(* CODESYS project AxisTest.project

Project tree, tasks and I/O mapping:
  Device : AC801-0221-U0R0, Shenzhen Inovance Technology Co., Ltd., version 3.5.11.50
    application Application
      libraries: Standard, * (System)
      task MainTask (cyclic, interval 4 ms, priority 2) calls nothing
      task ETHERCAT_C (cyclic, interval 4000 µs, priority 0) calls ETHERCAT_C.EtherCAT_Task, PLC_PRG
      program PLC_PRG [ST]
      DifferentialMonitor
      trace Trace (task ETHERCAT_C): PLC_PRG.adFbPos[0], PLC_PRG.adFbPos[1], PLC_PRG.adFbPos[2], PLC_PRG.adFbPos[3], PLC_PRG.lResult
      Symbols
    HardWare Configuration
    Network Configuration
      EtherCAT Config
    Device Diagnosis
    Resources List
    ConfigStorage
    SoftMotion General Axis Pool
    MODBUS_TCP : ModbusTCP本地从站, inovance, version 00.00.00.10
    HwConfiguratioinDevice : SystemConfig, Inovance, version 00.00.00.10
        settings: NetworkConfigArray.NetworkConfigArray.BusType = 10; NetworkConfigArray.NetworkConfigArray.RackSum = 1; NetworkConfigArray.NetworkConfigArray.HardwareConfigArray.HardwareConfigArray.RackNo = 1
    ETHERCAT_C : EtherCAT Master SoftMotion, 3S - Smart Software Solutions GmbH, version 3.5.11.10
        settings:  = 0; NetworkName = 'enp3s0'; SelectNetworkByName = TRUE; DisableTaskGeneration = True
      InoSV630N_3 : SV630_1Axis_03715, Inovance, order no. InoSV630N, version Revision=16#00010000
          settings: Number of Outputs = 6; Number of Inputs = 10; Number of Infos about Outputs = 6; Number of Infos about Inputs = 10; StationAlias = 0; Sync.Length = 18; Sync.Length = 32; FMMU.Length = 18; FMMU.Length = 32; AutoUpdate = False; DC sync0 cycletime = 4000; DC sync1 cycletime = 4000; Number of SDO = 10; Homing method.Index = 16#6098; Homing method.Subindex = 16#00; Homing method.Value = 1; Homing method.Size = 8; Homing method.AbortIfError = FALSE; Homing method.JumpToLine = FALSE; Homing method.Line = 0; Homing method.CompleteAccess = FALSE; Actual Position Calculation Method.Index = 16#60E6; Actual Position Calculation Method.Subindex = 16#00; Actual Position Calculation Method.Value = 0; Actual Position Calculation Method.Size = 8; Actual Position Calculation Method.AbortIfError = FALSE; Actual Position Calculation Method.JumpToLine = FALSE; Actual Position Calculation Method.Line = 0; Actual Position Calculation Method.CompleteAccess = FALSE; Speed during search for switch.Index = 16#6099; Speed during search for switch.Subindex = 16#01; Speed during search for switch.Value = 436907; Speed during search for switch.Size = 32; Speed during search for switch.AbortIfError = FALSE; Speed during search for switch.JumpToLine = FALSE; Speed during search for switch.Line = 0; Speed during search for switch.CompleteAccess = FALSE; Homing acceleration.Index = 16#609A; Homing acceleration.Subindex = 16#00; Homing acceleration.Value = 43690666;
            Homing acceleration.Size = 32; Homing acceleration.AbortIfError = FALSE; Homing acceleration.JumpToLine = FALSE; Homing acceleration.Line = 0; Homing acceleration.CompleteAccess = FALSE; Speed during search for zero.Index = 16#6099; Speed during search for zero.Subindex = 16#02; Speed during search for zero.Value = 43691; Speed during search for zero.Size = 32; Speed during search for zero.AbortIfError = FALSE; Speed during search for zero.JumpToLine = FALSE; Speed during search for zero.Line = 0; Speed during search for zero.CompleteAccess = FALSE; Time of home searching.Index = 16#2005; Time of home searching.Subindex = 16#24; Time of home searching.Value = 50000; Time of home searching.Size = 16; Time of home searching.AbortIfError = FALSE; Time of home searching.JumpToLine = FALSE; Time of home searching.Line = 0; Time of home searching.CompleteAccess = FALSE; Positive torque limit value.Index = 16#60E0; Positive torque limit value.Subindex = 16#00; Positive torque limit value.Value = 3500; Positive torque limit value.Size = 16; Positive torque limit value.AbortIfError = FALSE; Positive torque limit value.JumpToLine = FALSE; Positive torque limit value.Line = 0; Positive torque limit value.CompleteAccess = FALSE; Negative torque limit value.Index = 16#60E1; Negative torque limit value.Subindex = 16#00; Negative torque limit value.Value = 3500; Negative torque limit value.Size = 16; Negative torque limit value.AbortIfError = FALSE; Negative torque limit value.JumpToLine = FALSE; Negative torque limit value.Line = 0; Negative torque limit value.CompleteAccess = FALSE; Max profile velocity.Index = 16#607F; Max profile velocity.Subindex = 16#00; Max profile velocity.Value = 26214400;
            Max profile velocity.Size = 32; Max profile velocity.AbortIfError = FALSE; Max profile velocity.JumpToLine = FALSE; Max profile velocity.Line = 0; Max profile velocity.CompleteAccess = FALSE; RxTxPdo.NumberofEntries = 6; RxTxPdo.Sm = 2; Controlword.Index = 16#6040; Controlword.SubIndex = 0; Controlword.Size = 16; Controlword.DependOnSlot = false; Controlword.DependOnSlotGroup = false; Target position.Index = 16#607A; Target position.SubIndex = 0; Target position.Size = 32; Target position.DependOnSlot = false; Target position.DependOnSlotGroup = false; Touch probe function.Index = 16#60B8; Touch probe function.SubIndex = 0; Touch probe function.Size = 16; Touch probe function.DependOnSlot = false; Touch probe function.DependOnSlotGroup = false; Physical outputs.Index = 16#60FE; Physical outputs.SubIndex = 1; Physical outputs.Size = 32; Physical outputs.DependOnSlot = false; Physical outputs.DependOnSlotGroup = false; Target velocity.Index = 16#60FF; Target velocity.SubIndex = 0; Target velocity.Size = 32; Target velocity.DependOnSlot = false; Target velocity.DependOnSlotGroup = false; Target torque.Index = 16#6071; Target torque.SubIndex = 0; Target torque.Size = 16; Target torque.DependOnSlot = false; Target torque.DependOnSlotGroup = false; RxTxPdo.Sm = -1; RxTxPdo.NumberofEntries = 10; RxTxPdo.Sm = 3;
            Error code.Index = 16#603F; Error code.SubIndex = 0; Error code.Size = 16; Error code.DependOnSlot = false; Error code.DependOnSlotGroup = false; Statusword.Index = 16#6041; Statusword.SubIndex = 0; Statusword.Size = 16; Statusword.DependOnSlot = false; Statusword.DependOnSlotGroup = false; Position actual value.Index = 16#6064; Position actual value.SubIndex = 0; Position actual value.Size = 32; Position actual value.DependOnSlot = false; Position actual value.DependOnSlotGroup = false; Torque actual value.Index = 16#6077; Torque actual value.SubIndex = 0; Torque actual value.Size = 16; Torque actual value.DependOnSlot = false; Torque actual value.DependOnSlotGroup = false; Following error actual value.Index = 16#60F4; Following error actual value.SubIndex = 0; Following error actual value.Size = 32; Following error actual value.DependOnSlot = false; Following error actual value.DependOnSlotGroup = false; Touch probe status.Index = 16#60B9; Touch probe status.SubIndex = 0; Touch probe status.Size = 16; Touch probe status.DependOnSlot = false; Touch probe status.DependOnSlotGroup = false; Touch probe pos1 pos value.Index = 16#60BA; Touch probe pos1 pos value.SubIndex = 0; Touch probe pos1 pos value.Size = 32; Touch probe pos1 pos value.DependOnSlot = false; Touch probe pos1 pos value.DependOnSlotGroup = false; Touch probe pos2 pos value.Index = 16#60BC; Touch probe pos2 pos value.SubIndex = 0; Touch probe pos2 pos value.Size = 32; Touch probe pos2 pos value.DependOnSlot = false; Touch probe pos2 pos value.DependOnSlotGroup = false;
            Digital inputs.Index = 16#60FD; Digital inputs.SubIndex = 0; Digital inputs.Size = 32; Digital inputs.DependOnSlot = false; Digital inputs.DependOnSlotGroup = false; Velocity actual value.Index = 16#606C; Velocity actual value.SubIndex = 0; Velocity actual value.Size = 32; Velocity actual value.DependOnSlot = false; Velocity actual value.DependOnSlotGroup = false; RxTxPdo.Sm = -1; Controlword.Name = 'Controlword'; Controlword.DataType = 'UINT'; Target position.Name = 'Target position'; Target position.DataType = 'DINT'; Touch probe function.Name = 'Touch probe function'; Touch probe function.DataType = 'UINT'; Physical outputs.Name = 'Physical outputs'; Physical outputs.DataType = 'UDINT'; Target velocity.Name = 'Target velocity'; Target velocity.DataType = 'DINT'; Target torque.Name = 'Target torque'; Target torque.DataType = 'INT'; Error code.Name = 'Error code'; Error code.DataType = 'UINT'; Statusword.Name = 'Statusword'; Statusword.DataType = 'UINT'; Position actual value.Name = 'Position actual value'; Position actual value.DataType = 'DINT'; Torque actual value.Name = 'Torque actual value'; Torque actual value.DataType = 'INT'; Following error actual value.Name = 'Following error actual value'; Following error actual value.DataType = 'DINT'; Touch probe status.Name = 'Touch probe status'; Touch probe status.DataType = 'UINT'; Touch probe pos1 pos value.Name = 'Touch probe pos1 pos value'; Touch probe pos1 pos value.DataType = 'DINT'; Touch probe pos2 pos value.Name = 'Touch probe pos2 pos value'; Touch probe pos2 pos value.DataType = 'DINT'; Digital inputs.Name = 'Digital inputs';
            Digital inputs.DataType = 'UDINT'; Velocity actual value.Name = 'Velocity actual value'; Velocity actual value.DataType = 'DINT'
          output Application.PLC_PRG.adCmdPos[3] : DINT  // Target position
          input  Application.PLC_PRG.adFbPos[3] : DINT  // Position actual value
          unmapped channels: Controlword, Touch probe function, Physical outputs, Target velocity, Target torque, Error code, Statusword, Torque actual value, Following error actual value, Touch probe status, Touch probe pos1 pos value, Touch probe pos2 pos value, Digital inputs, Velocity actual value
        Axis_3 : Axis, Inovance, order no. 0, version 1.0.0.0
            settings: wDriveID = 3; dwRatioTechUnitsDenom = 262144; fSWMaxVelocity = 1000; fSWMaxAcceleration = 10000; fSWMaxDeceleration = 10000; fSWMaxJerk = 100000; iEncoderType = 1; iAbsEncoderOption = 1; HomingMode = 10; ZeroSignal = 0; StartDirction = 1; EndDirection = 1; PosLimitMode = 0; NegLimitMode = 0; HomingVelocity = 10; HomingApproachVelocity = 2; HomingAcceleration = 100; HomingDeceleration = 100; HomingJerk = 0; HomeMaskDistance = 0; HomePositionOffset = 0; HomePushTime = 0; HomeCompensation = 0; HomeTimeout = 0; HomeCompensationVelocity = 1000; 4000 = 0; 4001 = 0; 4003 = true; 4004 = 3; 4005 = 0; 4006 = 1.666667; 4007 = 166.666666; 4008 = 0.166667; 4009 = 50000; 4010 = 3500; 4011 = 3500; 4012 = 100.000000; ScalingIncs = 16#40000; 6005 = 1; AdrOffset_8010 = 72;
              BitOffset_8010 = 0; BitLength_8010 = 16; Address_8010 = '%QW36'; Type_8010 = 'UINT'; AddressPointer_8010 = ADR(%QW36); AdrOffset_8020 = 0; BitOffset_8020 = 0; BitLength_8020 = 32; Address_8020 = 'PLC_PRG.adCmdPos[3]'; Type_8020 = 'DINT'; AddressPointer_8020 = ADR(PLC_PRG.adCmdPos[3]); set velocity (diSetVelocity) = 1118; Object_8030 = 16#60FF:16#00; AdrOffset_8030 = 88; BitOffset_8030 = 0; BitLength_8030 = 32; Address_8030 = '%QD22'; Type_8030 = 'DINT'; AddressPointer_8030 = ADR(%QD22); set torque (wSetTorque) = 1168; Object_8040 = 16#6071:16#00; AdrOffset_8040 = 92; BitOffset_8040 = 0; BitLength_8040 = 16; Address_8040 = '%QW46'; Type_8040 = 'INT'; AddressPointer_8040 = ADR(%QW46); Modes of operation (OP) = 10096; Object_8050 = 16#6060:16#00; AdrOffset_8050 = 4294967295; BitOffset_8050 = 0; BitLength_8050 = 0; Address_8050 = ''; Type_8050 = ''; AddressPointer_8050 = 0; Touch Probe Function = 10184; Object_8060 = 16#60B8:16#00; AdrOffset_8060 = 80; BitOffset_8060 = 0; BitLength_8060 = 16;
              Address_8060 = '%QW40'; Type_8060 = 'UINT'; AddressPointer_8060 = ADR(%QW40); Add velocity value = 10177; Object_8070 = 16#60B1:16#00; AdrOffset_8070 = 4294967295; BitOffset_8070 = 0; BitLength_8070 = 0; Address_8070 = ''; Type_8070 = ''; AddressPointer_8070 = 0; Add torque value = 10178; Object_8080 = 16#60B2:16#00; AdrOffset_8080 = 4294967295; BitOffset_8080 = 0; BitLength_8080 = 0; Address_8080 = ''; Type_8080 = ''; AddressPointer_8080 = 0; Digital outputs (A637) = 10254; Object_8090 = 16#60FE:16#01; AdrOffset_8090 = 84; BitOffset_8090 = 0; BitLength_8090 = 32; Address_8090 = '%QD21'; Type_8090 = 'UDINT'; AddressPointer_8090 = ADR(%QD21); Max Profile Velocity = 2010; Object_8100 = 16#607F:16#00; AdrOffset_8100 = 4294967295; BitOffset_8100 = 0; BitLength_8100 = 0; Address_8100 = ''; Type_8100 = ''; AddressPointer_8100 = 0; AdrOffset_8510 = 110; BitOffset_8510 = 0; BitLength_8510 = 16; Address_8510 = '%IW55'; Type_8510 = 'UINT';
              AddressPointer_8510 = ADR(%IW55); AdrOffset_8520 = 0; BitOffset_8520 = 0; BitLength_8520 = 32; Address_8520 = 'PLC_PRG.adFbPos[3]'; Type_8520 = 'DINT'; AddressPointer_8520 = ADR(PLC_PRG.adFbPos[3]); actual velocity (diActVelocity) = 1119; Object_8530 = 16#606C:16#00; AdrOffset_8530 = 140; BitOffset_8530 = 0; BitLength_8530 = 32; Address_8530 = '%ID35'; Type_8530 = 'DINT'; AddressPointer_8530 = ADR(%ID35); actual torque (wActTorque) = 1169; Object_8540 = 16#6077:16#00; AdrOffset_8540 = 116; BitOffset_8540 = 0; BitLength_8540 = 16; Address_8540 = '%IW58'; Type_8540 = 'INT'; AddressPointer_8540 = ADR(%IW58); Modes of operation display (OP) = 20097; Object_8550 = 16#6061:16#00; AdrOffset_8550 = 4294967295; BitOffset_8550 = 0; BitLength_8550 = 0; Address_8550 = ''; Type_8550 = ''; AddressPointer_8550 = 0; digital inputs (in.dwDigitalInputs) = 20253; Object_8560 = 16#60FD:16#00; AdrOffset_8560 = 136; BitOffset_8560 = 0; BitLength_8560 = 32; Address_8560 = '%ID34'; Type_8560 = 'UDINT'; AddressPointer_8560 = ADR(%ID34); Touch Probe Status = 20185;
              Object_8570 = 16#60B9:16#00; AdrOffset_8570 = 124; BitOffset_8570 = 0; BitLength_8570 = 16; Address_8570 = '%IW62'; Type_8570 = 'UINT'; AddressPointer_8570 = ADR(%IW62); Touch Probe 1 rising edge = 20186; Object_8580 = 16#60BA:16#00; AdrOffset_8580 = 128; BitOffset_8580 = 0; BitLength_8580 = 32; Address_8580 = '%ID32'; Type_8580 = 'DINT'; AddressPointer_8580 = ADR(%ID32); Touch Probe 1 falling edge = 20187; Object_8590 = 16#60BB:16#00; AdrOffset_8590 = 4294967295; BitOffset_8590 = 0; BitLength_8590 = 0; Address_8590 = ''; Type_8590 = ''; AddressPointer_8590 = 0; Touch Probe 2 rising edge = 20188; Object_8600 = 16#60BC:16#00; AdrOffset_8600 = 132; BitOffset_8600 = 0; BitLength_8600 = 32; Address_8600 = '%ID33'; Type_8600 = 'DINT'; AddressPointer_8600 = ADR(%ID33); Touch Probe 2 falling edge = 20189; Object_8600 = 16#60BD:16#00; AdrOffset_8600 = 4294967295; BitOffset_8600 = 0; BitLength_8600 = 0; Address_8610 = ''; Type_8610 = ''; AddressPointer_8610 = 0; Error Code(603F) = 2020;
              Object_8620 = 16#603F:16#00; AdrOffset_8620 = 108; BitOffset_8620 = 0; BitLength_8620 = 16; Address_8620 = '%IW54'; Type_8620 = 'UINT'; AddressPointer_8620 = ADR(%IW54); Automatic Mapping = True; IsValid = True; IsHostHoming = False; PulseSelectIndex = 2
      InoSV630N_2 : SV630_1Axis_03715, Inovance, order no. InoSV630N, version Revision=16#00010000
          settings: Number of Outputs = 6; Number of Inputs = 10; Number of Infos about Outputs = 6; Number of Infos about Inputs = 10; StationAlias = 0; Sync.Length = 18; Sync.Length = 32; FMMU.Length = 18; FMMU.Length = 32; AutoUpdate = False; DC sync0 cycletime = 4000; DC sync1 cycletime = 4000; Number of SDO = 10; Homing method.Index = 16#6098; Homing method.Subindex = 16#00; Homing method.Value = 1; Homing method.Size = 8; Homing method.AbortIfError = FALSE; Homing method.JumpToLine = FALSE; Homing method.Line = 0; Homing method.CompleteAccess = FALSE; Actual Position Calculation Method.Index = 16#60E6; Actual Position Calculation Method.Subindex = 16#00; Actual Position Calculation Method.Value = 0; Actual Position Calculation Method.Size = 8; Actual Position Calculation Method.AbortIfError = FALSE; Actual Position Calculation Method.JumpToLine = FALSE; Actual Position Calculation Method.Line = 0; Actual Position Calculation Method.CompleteAccess = FALSE; Speed during search for switch.Index = 16#6099; Speed during search for switch.Subindex = 16#01; Speed during search for switch.Value = 436907; Speed during search for switch.Size = 32; Speed during search for switch.AbortIfError = FALSE; Speed during search for switch.JumpToLine = FALSE; Speed during search for switch.Line = 0; Speed during search for switch.CompleteAccess = FALSE; Homing acceleration.Index = 16#609A; Homing acceleration.Subindex = 16#00; Homing acceleration.Value = 43690666;
            Homing acceleration.Size = 32; Homing acceleration.AbortIfError = FALSE; Homing acceleration.JumpToLine = FALSE; Homing acceleration.Line = 0; Homing acceleration.CompleteAccess = FALSE; Speed during search for zero.Index = 16#6099; Speed during search for zero.Subindex = 16#02; Speed during search for zero.Value = 43691; Speed during search for zero.Size = 32; Speed during search for zero.AbortIfError = FALSE; Speed during search for zero.JumpToLine = FALSE; Speed during search for zero.Line = 0; Speed during search for zero.CompleteAccess = FALSE; Time of home searching.Index = 16#2005; Time of home searching.Subindex = 16#24; Time of home searching.Value = 50000; Time of home searching.Size = 16; Time of home searching.AbortIfError = FALSE; Time of home searching.JumpToLine = FALSE; Time of home searching.Line = 0; Time of home searching.CompleteAccess = FALSE; Positive torque limit value.Index = 16#60E0; Positive torque limit value.Subindex = 16#00; Positive torque limit value.Value = 3500; Positive torque limit value.Size = 16; Positive torque limit value.AbortIfError = FALSE; Positive torque limit value.JumpToLine = FALSE; Positive torque limit value.Line = 0; Positive torque limit value.CompleteAccess = FALSE; Negative torque limit value.Index = 16#60E1; Negative torque limit value.Subindex = 16#00; Negative torque limit value.Value = 3500; Negative torque limit value.Size = 16; Negative torque limit value.AbortIfError = FALSE; Negative torque limit value.JumpToLine = FALSE; Negative torque limit value.Line = 0; Negative torque limit value.CompleteAccess = FALSE; Max profile velocity.Index = 16#607F; Max profile velocity.Subindex = 16#00; Max profile velocity.Value = 26214400;
            Max profile velocity.Size = 32; Max profile velocity.AbortIfError = FALSE; Max profile velocity.JumpToLine = FALSE; Max profile velocity.Line = 0; Max profile velocity.CompleteAccess = FALSE; RxTxPdo.NumberofEntries = 6; RxTxPdo.Sm = 2; Controlword.Index = 16#6040; Controlword.SubIndex = 0; Controlword.Size = 16; Controlword.DependOnSlot = false; Controlword.DependOnSlotGroup = false; Target position.Index = 16#607A; Target position.SubIndex = 0; Target position.Size = 32; Target position.DependOnSlot = false; Target position.DependOnSlotGroup = false; Touch probe function.Index = 16#60B8; Touch probe function.SubIndex = 0; Touch probe function.Size = 16; Touch probe function.DependOnSlot = false; Touch probe function.DependOnSlotGroup = false; Physical outputs.Index = 16#60FE; Physical outputs.SubIndex = 1; Physical outputs.Size = 32; Physical outputs.DependOnSlot = false; Physical outputs.DependOnSlotGroup = false; Target velocity.Index = 16#60FF; Target velocity.SubIndex = 0; Target velocity.Size = 32; Target velocity.DependOnSlot = false; Target velocity.DependOnSlotGroup = false; Target torque.Index = 16#6071; Target torque.SubIndex = 0; Target torque.Size = 16; Target torque.DependOnSlot = false; Target torque.DependOnSlotGroup = false; RxTxPdo.Sm = -1; RxTxPdo.NumberofEntries = 10; RxTxPdo.Sm = 3;
            Error code.Index = 16#603F; Error code.SubIndex = 0; Error code.Size = 16; Error code.DependOnSlot = false; Error code.DependOnSlotGroup = false; Statusword.Index = 16#6041; Statusword.SubIndex = 0; Statusword.Size = 16; Statusword.DependOnSlot = false; Statusword.DependOnSlotGroup = false; Position actual value.Index = 16#6064; Position actual value.SubIndex = 0; Position actual value.Size = 32; Position actual value.DependOnSlot = false; Position actual value.DependOnSlotGroup = false; Torque actual value.Index = 16#6077; Torque actual value.SubIndex = 0; Torque actual value.Size = 16; Torque actual value.DependOnSlot = false; Torque actual value.DependOnSlotGroup = false; Following error actual value.Index = 16#60F4; Following error actual value.SubIndex = 0; Following error actual value.Size = 32; Following error actual value.DependOnSlot = false; Following error actual value.DependOnSlotGroup = false; Touch probe status.Index = 16#60B9; Touch probe status.SubIndex = 0; Touch probe status.Size = 16; Touch probe status.DependOnSlot = false; Touch probe status.DependOnSlotGroup = false; Touch probe pos1 pos value.Index = 16#60BA; Touch probe pos1 pos value.SubIndex = 0; Touch probe pos1 pos value.Size = 32; Touch probe pos1 pos value.DependOnSlot = false; Touch probe pos1 pos value.DependOnSlotGroup = false; Touch probe pos2 pos value.Index = 16#60BC; Touch probe pos2 pos value.SubIndex = 0; Touch probe pos2 pos value.Size = 32; Touch probe pos2 pos value.DependOnSlot = false; Touch probe pos2 pos value.DependOnSlotGroup = false;
            Digital inputs.Index = 16#60FD; Digital inputs.SubIndex = 0; Digital inputs.Size = 32; Digital inputs.DependOnSlot = false; Digital inputs.DependOnSlotGroup = false; Velocity actual value.Index = 16#606C; Velocity actual value.SubIndex = 0; Velocity actual value.Size = 32; Velocity actual value.DependOnSlot = false; Velocity actual value.DependOnSlotGroup = false; RxTxPdo.Sm = -1; Controlword.Name = 'Controlword'; Controlword.DataType = 'UINT'; Target position.Name = 'Target position'; Target position.DataType = 'DINT'; Touch probe function.Name = 'Touch probe function'; Touch probe function.DataType = 'UINT'; Physical outputs.Name = 'Physical outputs'; Physical outputs.DataType = 'UDINT'; Target velocity.Name = 'Target velocity'; Target velocity.DataType = 'DINT'; Target torque.Name = 'Target torque'; Target torque.DataType = 'INT'; Error code.Name = 'Error code'; Error code.DataType = 'UINT'; Statusword.Name = 'Statusword'; Statusword.DataType = 'UINT'; Position actual value.Name = 'Position actual value'; Position actual value.DataType = 'DINT'; Torque actual value.Name = 'Torque actual value'; Torque actual value.DataType = 'INT'; Following error actual value.Name = 'Following error actual value'; Following error actual value.DataType = 'DINT'; Touch probe status.Name = 'Touch probe status'; Touch probe status.DataType = 'UINT'; Touch probe pos1 pos value.Name = 'Touch probe pos1 pos value'; Touch probe pos1 pos value.DataType = 'DINT'; Touch probe pos2 pos value.Name = 'Touch probe pos2 pos value'; Touch probe pos2 pos value.DataType = 'DINT'; Digital inputs.Name = 'Digital inputs';
            Digital inputs.DataType = 'UDINT'; Velocity actual value.Name = 'Velocity actual value'; Velocity actual value.DataType = 'DINT'
          input  Application.PLC_PRG.adFbPos[2] : DINT  // Position actual value
          unmapped channels: Controlword, Target position, Touch probe function, Physical outputs, Target velocity, Target torque, Error code, Statusword, Torque actual value, Following error actual value, Touch probe status, Touch probe pos1 pos value, Touch probe pos2 pos value, Digital inputs, Velocity actual value
        Axis_2 : Axis, Inovance, order no. 0, version 1.0.0.0
            settings: wDriveID = 2; dwRatioTechUnitsDenom = 262144; fSWMaxVelocity = 1000; fSWMaxAcceleration = 10000; fSWMaxDeceleration = 10000; fSWMaxJerk = 100000; iEncoderType = 1; iAbsEncoderOption = 1; HomingMode = 10; ZeroSignal = 0; StartDirction = 1; EndDirection = 1; PosLimitMode = 0; NegLimitMode = 0; HomingVelocity = 10; HomingApproachVelocity = 2; HomingAcceleration = 100; HomingDeceleration = 100; HomingJerk = 0; HomeMaskDistance = 0; HomePositionOffset = 0; HomePushTime = 0; HomeCompensation = 0; HomeTimeout = 0; HomeCompensationVelocity = 1000; 4000 = 0; 4001 = 0; 4003 = true; 4004 = 3; 4005 = 0; 4006 = 1.666667; 4007 = 166.666666; 4008 = 0.166667; 4009 = 50000; 4010 = 3500; 4011 = 3500; 4012 = 100.000000; ScalingIncs = 16#40000; 6005 = 1; AdrOffset_8010 = 48;
              BitOffset_8010 = 0; BitLength_8010 = 16; Address_8010 = '%QW24'; Type_8010 = 'UINT'; AddressPointer_8010 = ADR(%QW24); AdrOffset_8020 = 52; BitOffset_8020 = 0; BitLength_8020 = 32; Address_8020 = '%QD13'; Type_8020 = 'DINT'; AddressPointer_8020 = ADR(%QD13); AdrOffset_8030 = 64; BitOffset_8030 = 0; BitLength_8030 = 32; Address_8030 = '%QD16'; Type_8030 = 'DINT'; AddressPointer_8030 = ADR(%QD16); AdrOffset_8040 = 68; BitOffset_8040 = 0; BitLength_8040 = 16; Address_8040 = '%QW34'; Type_8040 = 'INT'; AddressPointer_8040 = ADR(%QW34); AdrOffset_8050 = 4294967295; BitOffset_8050 = 0; BitLength_8050 = 0; Address_8050 = ''; Type_8050 = ''; AddressPointer_8050 = 0; AdrOffset_8060 = 56; BitOffset_8060 = 0; BitLength_8060 = 16; Address_8060 = '%QW28'; Type_8060 = 'UINT'; AddressPointer_8060 = ADR(%QW28); AdrOffset_8070 = 4294967295; BitOffset_8070 = 0; BitLength_8070 = 0; Address_8070 = ''; Type_8070 = '';
              AddressPointer_8070 = 0; AdrOffset_8080 = 4294967295; BitOffset_8080 = 0; BitLength_8080 = 0; Address_8080 = ''; Type_8080 = ''; AddressPointer_8080 = 0; AdrOffset_8090 = 60; BitOffset_8090 = 0; BitLength_8090 = 32; Address_8090 = '%QD15'; Type_8090 = 'UDINT'; AddressPointer_8090 = ADR(%QD15); AdrOffset_8100 = 4294967295; BitOffset_8100 = 0; BitLength_8100 = 0; Address_8100 = ''; Type_8100 = ''; AddressPointer_8100 = 0; AdrOffset_8510 = 74; BitOffset_8510 = 0; BitLength_8510 = 16; Address_8510 = '%IW37'; Type_8510 = 'UINT'; AddressPointer_8510 = ADR(%IW37); AdrOffset_8520 = 0; BitOffset_8520 = 0; BitLength_8520 = 32; Address_8520 = 'PLC_PRG.adFbPos[2]'; Type_8520 = 'DINT'; AddressPointer_8520 = ADR(PLC_PRG.adFbPos[2]); AdrOffset_8530 = 104; BitOffset_8530 = 0; BitLength_8530 = 32; Address_8530 = '%ID26'; Type_8530 = 'DINT'; AddressPointer_8530 = ADR(%ID26); AdrOffset_8540 = 80; BitOffset_8540 = 0; BitLength_8540 = 16;
              Address_8540 = '%IW40'; Type_8540 = 'INT'; AddressPointer_8540 = ADR(%IW40); AdrOffset_8550 = 4294967295; BitOffset_8550 = 0; BitLength_8550 = 0; Address_8550 = ''; Type_8550 = ''; AddressPointer_8550 = 0; AdrOffset_8560 = 100; BitOffset_8560 = 0; BitLength_8560 = 32; Address_8560 = '%ID25'; Type_8560 = 'UDINT'; AddressPointer_8560 = ADR(%ID25); AdrOffset_8570 = 88; BitOffset_8570 = 0; BitLength_8570 = 16; Address_8570 = '%IW44'; Type_8570 = 'UINT'; AddressPointer_8570 = ADR(%IW44); AdrOffset_8580 = 92; BitOffset_8580 = 0; BitLength_8580 = 32; Address_8580 = '%ID23'; Type_8580 = 'DINT'; AddressPointer_8580 = ADR(%ID23); AdrOffset_8590 = 4294967295; BitOffset_8590 = 0; BitLength_8590 = 0; Address_8590 = ''; Type_8590 = ''; AddressPointer_8590 = 0; AdrOffset_8600 = 96; BitOffset_8600 = 0; BitLength_8600 = 32; Address_8600 = '%ID24'; Type_8600 = 'DINT'; AddressPointer_8600 = ADR(%ID24); AdrOffset_8600 = 4294967295;
              BitOffset_8600 = 0; BitLength_8600 = 0; Address_8610 = ''; Type_8610 = ''; AddressPointer_8610 = 0; AdrOffset_8620 = 72; BitOffset_8620 = 0; BitLength_8620 = 16; Address_8620 = '%IW36'; Type_8620 = 'UINT'; AddressPointer_8620 = ADR(%IW36); IsValid = True; IsHostHoming = False; PulseSelectIndex = 2
      InoSV630N_1 : SV630_1Axis_03715, Inovance, order no. InoSV630N, version Revision=16#00010000
          settings: Number of Outputs = 6; Number of Inputs = 10; Number of Infos about Outputs = 6; Number of Infos about Inputs = 10; StationAlias = 0; Sync.Length = 18; Sync.Length = 32; FMMU.Length = 18; FMMU.Length = 32; AutoUpdate = False; DC sync0 cycletime = 4000; DC sync1 cycletime = 4000; Number of SDO = 10; Homing method.Index = 16#6098; Homing method.Subindex = 16#00; Homing method.Value = 1; Homing method.Size = 8; Homing method.AbortIfError = FALSE; Homing method.JumpToLine = FALSE; Homing method.Line = 0; Homing method.CompleteAccess = FALSE; Actual Position Calculation Method.Index = 16#60E6; Actual Position Calculation Method.Subindex = 16#00; Actual Position Calculation Method.Value = 0; Actual Position Calculation Method.Size = 8; Actual Position Calculation Method.AbortIfError = FALSE; Actual Position Calculation Method.JumpToLine = FALSE; Actual Position Calculation Method.Line = 0; Actual Position Calculation Method.CompleteAccess = FALSE; Speed during search for switch.Index = 16#6099; Speed during search for switch.Subindex = 16#01; Speed during search for switch.Value = 436907; Speed during search for switch.Size = 32; Speed during search for switch.AbortIfError = FALSE; Speed during search for switch.JumpToLine = FALSE; Speed during search for switch.Line = 0; Speed during search for switch.CompleteAccess = FALSE; Homing acceleration.Index = 16#609A; Homing acceleration.Subindex = 16#00; Homing acceleration.Value = 43690666;
            Homing acceleration.Size = 32; Homing acceleration.AbortIfError = FALSE; Homing acceleration.JumpToLine = FALSE; Homing acceleration.Line = 0; Homing acceleration.CompleteAccess = FALSE; Speed during search for zero.Index = 16#6099; Speed during search for zero.Subindex = 16#02; Speed during search for zero.Value = 43691; Speed during search for zero.Size = 32; Speed during search for zero.AbortIfError = FALSE; Speed during search for zero.JumpToLine = FALSE; Speed during search for zero.Line = 0; Speed during search for zero.CompleteAccess = FALSE; Time of home searching.Index = 16#2005; Time of home searching.Subindex = 16#24; Time of home searching.Value = 50000; Time of home searching.Size = 16; Time of home searching.AbortIfError = FALSE; Time of home searching.JumpToLine = FALSE; Time of home searching.Line = 0; Time of home searching.CompleteAccess = FALSE; Positive torque limit value.Index = 16#60E0; Positive torque limit value.Subindex = 16#00; Positive torque limit value.Value = 3500; Positive torque limit value.Size = 16; Positive torque limit value.AbortIfError = FALSE; Positive torque limit value.JumpToLine = FALSE; Positive torque limit value.Line = 0; Positive torque limit value.CompleteAccess = FALSE; Negative torque limit value.Index = 16#60E1; Negative torque limit value.Subindex = 16#00; Negative torque limit value.Value = 3500; Negative torque limit value.Size = 16; Negative torque limit value.AbortIfError = FALSE; Negative torque limit value.JumpToLine = FALSE; Negative torque limit value.Line = 0; Negative torque limit value.CompleteAccess = FALSE; Max profile velocity.Index = 16#607F; Max profile velocity.Subindex = 16#00; Max profile velocity.Value = 26214400;
            Max profile velocity.Size = 32; Max profile velocity.AbortIfError = FALSE; Max profile velocity.JumpToLine = FALSE; Max profile velocity.Line = 0; Max profile velocity.CompleteAccess = FALSE; RxTxPdo.NumberofEntries = 6; RxTxPdo.Sm = 2; Controlword.Index = 16#6040; Controlword.SubIndex = 0; Controlword.Size = 16; Controlword.DependOnSlot = false; Controlword.DependOnSlotGroup = false; Target position.Index = 16#607A; Target position.SubIndex = 0; Target position.Size = 32; Target position.DependOnSlot = false; Target position.DependOnSlotGroup = false; Touch probe function.Index = 16#60B8; Touch probe function.SubIndex = 0; Touch probe function.Size = 16; Touch probe function.DependOnSlot = false; Touch probe function.DependOnSlotGroup = false; Physical outputs.Index = 16#60FE; Physical outputs.SubIndex = 1; Physical outputs.Size = 32; Physical outputs.DependOnSlot = false; Physical outputs.DependOnSlotGroup = false; Target velocity.Index = 16#60FF; Target velocity.SubIndex = 0; Target velocity.Size = 32; Target velocity.DependOnSlot = false; Target velocity.DependOnSlotGroup = false; Target torque.Index = 16#6071; Target torque.SubIndex = 0; Target torque.Size = 16; Target torque.DependOnSlot = false; Target torque.DependOnSlotGroup = false; RxTxPdo.Sm = -1; RxTxPdo.NumberofEntries = 10; RxTxPdo.Sm = 3;
            Error code.Index = 16#603F; Error code.SubIndex = 0; Error code.Size = 16; Error code.DependOnSlot = false; Error code.DependOnSlotGroup = false; Statusword.Index = 16#6041; Statusword.SubIndex = 0; Statusword.Size = 16; Statusword.DependOnSlot = false; Statusword.DependOnSlotGroup = false; Position actual value.Index = 16#6064; Position actual value.SubIndex = 0; Position actual value.Size = 32; Position actual value.DependOnSlot = false; Position actual value.DependOnSlotGroup = false; Torque actual value.Index = 16#6077; Torque actual value.SubIndex = 0; Torque actual value.Size = 16; Torque actual value.DependOnSlot = false; Torque actual value.DependOnSlotGroup = false; Following error actual value.Index = 16#60F4; Following error actual value.SubIndex = 0; Following error actual value.Size = 32; Following error actual value.DependOnSlot = false; Following error actual value.DependOnSlotGroup = false; Touch probe status.Index = 16#60B9; Touch probe status.SubIndex = 0; Touch probe status.Size = 16; Touch probe status.DependOnSlot = false; Touch probe status.DependOnSlotGroup = false; Touch probe pos1 pos value.Index = 16#60BA; Touch probe pos1 pos value.SubIndex = 0; Touch probe pos1 pos value.Size = 32; Touch probe pos1 pos value.DependOnSlot = false; Touch probe pos1 pos value.DependOnSlotGroup = false; Touch probe pos2 pos value.Index = 16#60BC; Touch probe pos2 pos value.SubIndex = 0; Touch probe pos2 pos value.Size = 32; Touch probe pos2 pos value.DependOnSlot = false; Touch probe pos2 pos value.DependOnSlotGroup = false;
            Digital inputs.Index = 16#60FD; Digital inputs.SubIndex = 0; Digital inputs.Size = 32; Digital inputs.DependOnSlot = false; Digital inputs.DependOnSlotGroup = false; Velocity actual value.Index = 16#606C; Velocity actual value.SubIndex = 0; Velocity actual value.Size = 32; Velocity actual value.DependOnSlot = false; Velocity actual value.DependOnSlotGroup = false; RxTxPdo.Sm = -1; Controlword.Name = 'Controlword'; Controlword.DataType = 'UINT'; Target position.Name = 'Target position'; Target position.DataType = 'DINT'; Touch probe function.Name = 'Touch probe function'; Touch probe function.DataType = 'UINT'; Physical outputs.Name = 'Physical outputs'; Physical outputs.DataType = 'UDINT'; Target velocity.Name = 'Target velocity'; Target velocity.DataType = 'DINT'; Target torque.Name = 'Target torque'; Target torque.DataType = 'INT'; Error code.Name = 'Error code'; Error code.DataType = 'UINT'; Statusword.Name = 'Statusword'; Statusword.DataType = 'UINT'; Position actual value.Name = 'Position actual value'; Position actual value.DataType = 'DINT'; Torque actual value.Name = 'Torque actual value'; Torque actual value.DataType = 'INT'; Following error actual value.Name = 'Following error actual value'; Following error actual value.DataType = 'DINT'; Touch probe status.Name = 'Touch probe status'; Touch probe status.DataType = 'UINT'; Touch probe pos1 pos value.Name = 'Touch probe pos1 pos value'; Touch probe pos1 pos value.DataType = 'DINT'; Touch probe pos2 pos value.Name = 'Touch probe pos2 pos value'; Touch probe pos2 pos value.DataType = 'DINT'; Digital inputs.Name = 'Digital inputs';
            Digital inputs.DataType = 'UDINT'; Velocity actual value.Name = 'Velocity actual value'; Velocity actual value.DataType = 'DINT'
          input  Application.PLC_PRG.adFbPos[1] : DINT  // Position actual value
          unmapped channels: Controlword, Target position, Touch probe function, Physical outputs, Target velocity, Target torque, Error code, Statusword, Torque actual value, Following error actual value, Touch probe status, Touch probe pos1 pos value, Touch probe pos2 pos value, Digital inputs, Velocity actual value
        Axis_1 : Axis, Inovance, order no. 0, version 1.0.0.0
            settings: dwRatioTechUnitsDenom = 262144; fSWMaxVelocity = 1000; fSWMaxAcceleration = 10000; fSWMaxDeceleration = 10000; fSWMaxJerk = 100000; iEncoderType = 1; iAbsEncoderOption = 1; HomingMode = 10; ZeroSignal = 0; StartDirction = 1; EndDirection = 1; PosLimitMode = 0; NegLimitMode = 0; HomingVelocity = 10; HomingApproachVelocity = 2; HomingAcceleration = 100; HomingDeceleration = 100; HomingJerk = 0; HomeMaskDistance = 0; HomePositionOffset = 0; HomePushTime = 0; HomeCompensation = 0; HomeTimeout = 0; HomeCompensationVelocity = 1000; 4000 = 0; 4001 = 0; 4003 = true; 4004 = 3; 4005 = 0; 4006 = 1.666667; 4007 = 166.666666; 4008 = 0.166667; 4009 = 50000; 4010 = 3500; 4011 = 3500; 4012 = 100.000000; ScalingIncs = 16#40000; 6005 = 1; AdrOffset_8010 = 24; BitOffset_8010 = 0;
              BitLength_8010 = 16; Address_8010 = '%QW12'; Type_8010 = 'UINT'; AddressPointer_8010 = ADR(%QW12); AdrOffset_8020 = 28; BitOffset_8020 = 0; BitLength_8020 = 32; Address_8020 = '%QD7'; Type_8020 = 'DINT'; AddressPointer_8020 = ADR(%QD7); AdrOffset_8030 = 40; BitOffset_8030 = 0; BitLength_8030 = 32; Address_8030 = '%QD10'; Type_8030 = 'DINT'; AddressPointer_8030 = ADR(%QD10); AdrOffset_8040 = 44; BitOffset_8040 = 0; BitLength_8040 = 16; Address_8040 = '%QW22'; Type_8040 = 'INT'; AddressPointer_8040 = ADR(%QW22); AdrOffset_8050 = 4294967295; BitOffset_8050 = 0; BitLength_8050 = 0; Address_8050 = ''; Type_8050 = ''; AddressPointer_8050 = 0; AdrOffset_8060 = 32; BitOffset_8060 = 0; BitLength_8060 = 16; Address_8060 = '%QW16'; Type_8060 = 'UINT'; AddressPointer_8060 = ADR(%QW16); AdrOffset_8070 = 4294967295; BitOffset_8070 = 0; BitLength_8070 = 0; Address_8070 = ''; Type_8070 = ''; AddressPointer_8070 = 0;
              AdrOffset_8080 = 4294967295; BitOffset_8080 = 0; BitLength_8080 = 0; Address_8080 = ''; Type_8080 = ''; AddressPointer_8080 = 0; AdrOffset_8090 = 36; BitOffset_8090 = 0; BitLength_8090 = 32; Address_8090 = '%QD9'; Type_8090 = 'UDINT'; AddressPointer_8090 = ADR(%QD9); AdrOffset_8100 = 4294967295; BitOffset_8100 = 0; BitLength_8100 = 0; Address_8100 = ''; Type_8100 = ''; AddressPointer_8100 = 0; AdrOffset_8510 = 38; BitOffset_8510 = 0; BitLength_8510 = 16; Address_8510 = '%IW19'; Type_8510 = 'UINT'; AddressPointer_8510 = ADR(%IW19); AdrOffset_8520 = 0; BitOffset_8520 = 0; BitLength_8520 = 32; Address_8520 = 'PLC_PRG.adFbPos[1]'; Type_8520 = 'DINT'; AddressPointer_8520 = ADR(PLC_PRG.adFbPos[1]); AdrOffset_8530 = 68; BitOffset_8530 = 0; BitLength_8530 = 32; Address_8530 = '%ID17'; Type_8530 = 'DINT'; AddressPointer_8530 = ADR(%ID17); AdrOffset_8540 = 44; BitOffset_8540 = 0; BitLength_8540 = 16; Address_8540 = '%IW22';
              Type_8540 = 'INT'; AddressPointer_8540 = ADR(%IW22); AdrOffset_8550 = 4294967295; BitOffset_8550 = 0; BitLength_8550 = 0; Address_8550 = ''; Type_8550 = ''; AddressPointer_8550 = 0; AdrOffset_8560 = 64; BitOffset_8560 = 0; BitLength_8560 = 32; Address_8560 = '%ID16'; Type_8560 = 'UDINT'; AddressPointer_8560 = ADR(%ID16); AdrOffset_8570 = 52; BitOffset_8570 = 0; BitLength_8570 = 16; Address_8570 = '%IW26'; Type_8570 = 'UINT'; AddressPointer_8570 = ADR(%IW26); AdrOffset_8580 = 56; BitOffset_8580 = 0; BitLength_8580 = 32; Address_8580 = '%ID14'; Type_8580 = 'DINT'; AddressPointer_8580 = ADR(%ID14); AdrOffset_8590 = 4294967295; BitOffset_8590 = 0; BitLength_8590 = 0; Address_8590 = ''; Type_8590 = ''; AddressPointer_8590 = 0; AdrOffset_8600 = 60; BitOffset_8600 = 0; BitLength_8600 = 32; Address_8600 = '%ID15'; Type_8600 = 'DINT'; AddressPointer_8600 = ADR(%ID15); AdrOffset_8600 = 4294967295; BitOffset_8600 = 0;
              BitLength_8600 = 0; Address_8610 = ''; Type_8610 = ''; AddressPointer_8610 = 0; AdrOffset_8620 = 36; BitOffset_8620 = 0; BitLength_8620 = 16; Address_8620 = '%IW18'; Type_8620 = 'UINT'; AddressPointer_8620 = ADR(%IW18); IsValid = True; IsHostHoming = False; PulseSelectIndex = 2
      InoSV630N : SV630_1Axis_03715, Inovance, order no. InoSV630N, version Revision=16#00010000
          settings: Number of Outputs = 6; Number of Inputs = 10; Number of Infos about Outputs = 6; Number of Infos about Inputs = 10; StationAlias = 0; Sync.Length = 18; Sync.Length = 32; FMMU.Length = 18; FMMU.Length = 32; AutoUpdate = False; DC sync0 cycletime = 4000; DC sync1 cycletime = 4000; Number of SDO = 10; Homing method.Index = 16#6098; Homing method.Subindex = 16#00; Homing method.Value = 1; Homing method.Size = 8; Homing method.AbortIfError = FALSE; Homing method.JumpToLine = FALSE; Homing method.Line = 0; Homing method.CompleteAccess = FALSE; Actual Position Calculation Method.Index = 16#60E6; Actual Position Calculation Method.Subindex = 16#00; Actual Position Calculation Method.Value = 0; Actual Position Calculation Method.Size = 8; Actual Position Calculation Method.AbortIfError = FALSE; Actual Position Calculation Method.JumpToLine = FALSE; Actual Position Calculation Method.Line = 0; Actual Position Calculation Method.CompleteAccess = FALSE; Speed during search for switch.Index = 16#6099; Speed during search for switch.Subindex = 16#01; Speed during search for switch.Value = 436907; Speed during search for switch.Size = 32; Speed during search for switch.AbortIfError = FALSE; Speed during search for switch.JumpToLine = FALSE; Speed during search for switch.Line = 0; Speed during search for switch.CompleteAccess = FALSE; Homing acceleration.Index = 16#609A; Homing acceleration.Subindex = 16#00; Homing acceleration.Value = 43690666;
            Homing acceleration.Size = 32; Homing acceleration.AbortIfError = FALSE; Homing acceleration.JumpToLine = FALSE; Homing acceleration.Line = 0; Homing acceleration.CompleteAccess = FALSE; Speed during search for zero.Index = 16#6099; Speed during search for zero.Subindex = 16#02; Speed during search for zero.Value = 43691; Speed during search for zero.Size = 32; Speed during search for zero.AbortIfError = FALSE; Speed during search for zero.JumpToLine = FALSE; Speed during search for zero.Line = 0; Speed during search for zero.CompleteAccess = FALSE; Time of home searching.Index = 16#2005; Time of home searching.Subindex = 16#24; Time of home searching.Value = 50000; Time of home searching.Size = 16; Time of home searching.AbortIfError = FALSE; Time of home searching.JumpToLine = FALSE; Time of home searching.Line = 0; Time of home searching.CompleteAccess = FALSE; Positive torque limit value.Index = 16#60E0; Positive torque limit value.Subindex = 16#00; Positive torque limit value.Value = 3500; Positive torque limit value.Size = 16; Positive torque limit value.AbortIfError = FALSE; Positive torque limit value.JumpToLine = FALSE; Positive torque limit value.Line = 0; Positive torque limit value.CompleteAccess = FALSE; Negative torque limit value.Index = 16#60E1; Negative torque limit value.Subindex = 16#00; Negative torque limit value.Value = 3500; Negative torque limit value.Size = 16; Negative torque limit value.AbortIfError = FALSE; Negative torque limit value.JumpToLine = FALSE; Negative torque limit value.Line = 0; Negative torque limit value.CompleteAccess = FALSE; Max profile velocity.Index = 16#607F; Max profile velocity.Subindex = 16#00; Max profile velocity.Value = 26214400;
            Max profile velocity.Size = 32; Max profile velocity.AbortIfError = FALSE; Max profile velocity.JumpToLine = FALSE; Max profile velocity.Line = 0; Max profile velocity.CompleteAccess = FALSE; RxTxPdo.NumberofEntries = 6; RxTxPdo.Sm = 2; Controlword.Index = 16#6040; Controlword.SubIndex = 0; Controlword.Size = 16; Controlword.DependOnSlot = false; Controlword.DependOnSlotGroup = false; Target position.Index = 16#607A; Target position.SubIndex = 0; Target position.Size = 32; Target position.DependOnSlot = false; Target position.DependOnSlotGroup = false; Touch probe function.Index = 16#60B8; Touch probe function.SubIndex = 0; Touch probe function.Size = 16; Touch probe function.DependOnSlot = false; Touch probe function.DependOnSlotGroup = false; Physical outputs.Index = 16#60FE; Physical outputs.SubIndex = 1; Physical outputs.Size = 32; Physical outputs.DependOnSlot = false; Physical outputs.DependOnSlotGroup = false; Target velocity.Index = 16#60FF; Target velocity.SubIndex = 0; Target velocity.Size = 32; Target velocity.DependOnSlot = false; Target velocity.DependOnSlotGroup = false; Target torque.Index = 16#6071; Target torque.SubIndex = 0; Target torque.Size = 16; Target torque.DependOnSlot = false; Target torque.DependOnSlotGroup = false; RxTxPdo.Sm = -1; RxTxPdo.NumberofEntries = 10; RxTxPdo.Sm = 3;
            Error code.Index = 16#603F; Error code.SubIndex = 0; Error code.Size = 16; Error code.DependOnSlot = false; Error code.DependOnSlotGroup = false; Statusword.Index = 16#6041; Statusword.SubIndex = 0; Statusword.Size = 16; Statusword.DependOnSlot = false; Statusword.DependOnSlotGroup = false; Position actual value.Index = 16#6064; Position actual value.SubIndex = 0; Position actual value.Size = 32; Position actual value.DependOnSlot = false; Position actual value.DependOnSlotGroup = false; Torque actual value.Index = 16#6077; Torque actual value.SubIndex = 0; Torque actual value.Size = 16; Torque actual value.DependOnSlot = false; Torque actual value.DependOnSlotGroup = false; Following error actual value.Index = 16#60F4; Following error actual value.SubIndex = 0; Following error actual value.Size = 32; Following error actual value.DependOnSlot = false; Following error actual value.DependOnSlotGroup = false; Touch probe status.Index = 16#60B9; Touch probe status.SubIndex = 0; Touch probe status.Size = 16; Touch probe status.DependOnSlot = false; Touch probe status.DependOnSlotGroup = false; Touch probe pos1 pos value.Index = 16#60BA; Touch probe pos1 pos value.SubIndex = 0; Touch probe pos1 pos value.Size = 32; Touch probe pos1 pos value.DependOnSlot = false; Touch probe pos1 pos value.DependOnSlotGroup = false; Touch probe pos2 pos value.Index = 16#60BC; Touch probe pos2 pos value.SubIndex = 0; Touch probe pos2 pos value.Size = 32; Touch probe pos2 pos value.DependOnSlot = false; Touch probe pos2 pos value.DependOnSlotGroup = false;
            Digital inputs.Index = 16#60FD; Digital inputs.SubIndex = 0; Digital inputs.Size = 32; Digital inputs.DependOnSlot = false; Digital inputs.DependOnSlotGroup = false; Velocity actual value.Index = 16#606C; Velocity actual value.SubIndex = 0; Velocity actual value.Size = 32; Velocity actual value.DependOnSlot = false; Velocity actual value.DependOnSlotGroup = false; RxTxPdo.Sm = -1; Controlword.Name = 'Controlword'; Controlword.DataType = 'UINT'; Target position.Name = 'Target position'; Target position.DataType = 'DINT'; Touch probe function.Name = 'Touch probe function'; Touch probe function.DataType = 'UINT'; Physical outputs.Name = 'Physical outputs'; Physical outputs.DataType = 'UDINT'; Target velocity.Name = 'Target velocity'; Target velocity.DataType = 'DINT'; Target torque.Name = 'Target torque'; Target torque.DataType = 'INT'; Error code.Name = 'Error code'; Error code.DataType = 'UINT'; Statusword.Name = 'Statusword'; Statusword.DataType = 'UINT'; Position actual value.Name = 'Position actual value'; Position actual value.DataType = 'DINT'; Torque actual value.Name = 'Torque actual value'; Torque actual value.DataType = 'INT'; Following error actual value.Name = 'Following error actual value'; Following error actual value.DataType = 'DINT'; Touch probe status.Name = 'Touch probe status'; Touch probe status.DataType = 'UINT'; Touch probe pos1 pos value.Name = 'Touch probe pos1 pos value'; Touch probe pos1 pos value.DataType = 'DINT'; Touch probe pos2 pos value.Name = 'Touch probe pos2 pos value'; Touch probe pos2 pos value.DataType = 'DINT'; Digital inputs.Name = 'Digital inputs';
            Digital inputs.DataType = 'UDINT'; Velocity actual value.Name = 'Velocity actual value'; Velocity actual value.DataType = 'DINT'
          input  Application.PLC_PRG.adFbPos[0] : DINT  // Position actual value
          unmapped channels: Controlword, Target position, Touch probe function, Physical outputs, Target velocity, Target torque, Error code, Statusword, Torque actual value, Following error actual value, Touch probe status, Touch probe pos1 pos value, Touch probe pos2 pos value, Digital inputs, Velocity actual value
        Axis_0 : Axis, Inovance, order no. 0, version 1.0.0.0
            settings: wDriveID = 0; dwRatioTechUnitsDenom = 262144; fSWMaxVelocity = 1000; fSWMaxAcceleration = 10000; fSWMaxDeceleration = 10000; fSWMaxJerk = 100000; iEncoderType = 1; iAbsEncoderOption = 1; HomingMode = 10; ZeroSignal = 0; StartDirction = 1; EndDirection = 1; PosLimitMode = 0; NegLimitMode = 0; HomingVelocity = 10; HomingApproachVelocity = 2; HomingAcceleration = 100; HomingDeceleration = 100; HomingJerk = 0; HomeMaskDistance = 0; HomePositionOffset = 0; HomePushTime = 0; HomeCompensation = 0; HomeTimeout = 0; HomeCompensationVelocity = 1000; 4000 = 0; 4001 = 0; 4003 = true; 4004 = 3; 4005 = 0; 4006 = 1.666667; 4007 = 166.666666; 4008 = 0.166667; 4009 = 50000; 4010 = 3500; 4011 = 3500; 4012 = 100.000000; ScalingIncs = 16#40000; 6005 = 1; AdrOffset_8010 = 0;
              BitOffset_8010 = 0; BitLength_8010 = 16; Address_8010 = '%QW0'; Type_8010 = 'UINT'; AddressPointer_8010 = ADR(%QW0); AdrOffset_8020 = 4; BitOffset_8020 = 0; BitLength_8020 = 32; Address_8020 = '%QD1'; Type_8020 = 'DINT'; AddressPointer_8020 = ADR(%QD1); AdrOffset_8030 = 16; BitOffset_8030 = 0; BitLength_8030 = 32; Address_8030 = '%QD4'; Type_8030 = 'DINT'; AddressPointer_8030 = ADR(%QD4); AdrOffset_8040 = 20; BitOffset_8040 = 0; BitLength_8040 = 16; Address_8040 = '%QW10'; Type_8040 = 'INT'; AddressPointer_8040 = ADR(%QW10); AdrOffset_8050 = 4294967295; BitOffset_8050 = 0; BitLength_8050 = 0; Address_8050 = ''; Type_8050 = ''; AddressPointer_8050 = 0; AdrOffset_8060 = 8; BitOffset_8060 = 0; BitLength_8060 = 16; Address_8060 = '%QW4'; Type_8060 = 'UINT'; AddressPointer_8060 = ADR(%QW4); AdrOffset_8070 = 4294967295; BitOffset_8070 = 0; BitLength_8070 = 0; Address_8070 = ''; Type_8070 = '';
              AddressPointer_8070 = 0; AdrOffset_8080 = 4294967295; BitOffset_8080 = 0; BitLength_8080 = 0; Address_8080 = ''; Type_8080 = ''; AddressPointer_8080 = 0; AdrOffset_8090 = 12; BitOffset_8090 = 0; BitLength_8090 = 32; Address_8090 = '%QD3'; Type_8090 = 'UDINT'; AddressPointer_8090 = ADR(%QD3); AdrOffset_8100 = 4294967295; BitOffset_8100 = 0; BitLength_8100 = 0; Address_8100 = ''; Type_8100 = ''; AddressPointer_8100 = 0; AdrOffset_8510 = 2; BitOffset_8510 = 0; BitLength_8510 = 16; Address_8510 = '%IW1'; Type_8510 = 'UINT'; AddressPointer_8510 = ADR(%IW1); AdrOffset_8520 = 0; BitOffset_8520 = 0; BitLength_8520 = 32; Address_8520 = 'PLC_PRG.adFbPos[0]'; Type_8520 = 'DINT'; AddressPointer_8520 = ADR(PLC_PRG.adFbPos[0]); AdrOffset_8530 = 32; BitOffset_8530 = 0; BitLength_8530 = 32; Address_8530 = '%ID8'; Type_8530 = 'DINT'; AddressPointer_8530 = ADR(%ID8); AdrOffset_8540 = 8; BitOffset_8540 = 0; BitLength_8540 = 16;
              Address_8540 = '%IW4'; Type_8540 = 'INT'; AddressPointer_8540 = ADR(%IW4); AdrOffset_8550 = 4294967295; BitOffset_8550 = 0; BitLength_8550 = 0; Address_8550 = ''; Type_8550 = ''; AddressPointer_8550 = 0; AdrOffset_8560 = 28; BitOffset_8560 = 0; BitLength_8560 = 32; Address_8560 = '%ID7'; Type_8560 = 'UDINT'; AddressPointer_8560 = ADR(%ID7); AdrOffset_8570 = 16; BitOffset_8570 = 0; BitLength_8570 = 16; Address_8570 = '%IW8'; Type_8570 = 'UINT'; AddressPointer_8570 = ADR(%IW8); AdrOffset_8580 = 20; BitOffset_8580 = 0; BitLength_8580 = 32; Address_8580 = '%ID5'; Type_8580 = 'DINT'; AddressPointer_8580 = ADR(%ID5); AdrOffset_8590 = 4294967295; BitOffset_8590 = 0; BitLength_8590 = 0; Address_8590 = ''; Type_8590 = ''; AddressPointer_8590 = 0; AdrOffset_8600 = 24; BitOffset_8600 = 0; BitLength_8600 = 32; Address_8600 = '%ID6'; Type_8600 = 'DINT'; AddressPointer_8600 = ADR(%ID6); AdrOffset_8600 = 4294967295;
              BitOffset_8600 = 0; BitLength_8600 = 0; Address_8610 = ''; Type_8610 = ''; AddressPointer_8610 = 0; AdrOffset_8620 = 0; BitOffset_8620 = 0; BitLength_8620 = 16; Address_8620 = '%IW0'; Type_8620 = 'UINT'; AddressPointer_8620 = ADR(%IW0); IsValid = True; IsHostHoming = False; PulseSelectIndex = 2
*)

// Device/Application/PLC_PRG
PROGRAM PLC_PRG
VAR
	iCounter	: INT := 0;
	iAxisNum	: INT := 0;
	bMoveStatus	: INT := 2;
	iVel		: INT := 2;
	bFirstRun	: BOOL := TRUE;
	bEnable	    : BOOL := FALSE;
	bReset	    : BOOL := FALSE;
	bForward	: BOOL := FALSE;
	bBackward	: BOOL := FALSE;
	bMoveTo		: BOOL := FALSE;
	bMoveToLen	: INT := 3;
	bMoveToDone	: BOOL := FALSE;
	bContinusMove	: BOOL := FALSE;
	bSingleAxisMove	: BOOL := FALSE;
	
	bSinMove    : BOOL := FALSE;
	dSinAmpl	: LREAL := 0.01;  // 振幅
	lSinFreq    : LREAL := 1;	  // 频率
	lSinFreqStep: LREAL := 3.0;
	lResult     : LREAL;
	adFbPos     : ARRAY[0..3] OF DINT;
	adFbForce    : ARRAY[0..3] OF INT;
	adFbPosTest     : ARRAY[0..3] OF LREAL;
	adCmdPos    : ARRAY[0..3] OF DINT;
	
	apMC_Jog    : ARRAY[0..3] OF MC_Jog;
	apMC_Power  : ARRAY[0..3] OF MC_Power;
	apAxis      : ARRAY[0..3] OF POINTER TO AXIS_REF_SM3;//定义轴
	apMC_MoveAbsolute : ARRAY[0..3] OF MC_MoveAbsolute;	//功能块声明
	apMC_Reset  : ARRAY[0..3] OF MC_Reset;
END_VAR


IF bFirstRun THEN
	apAxis[0] := ADR(Axis_0);
	apAxis[1] := ADR(Axis_1);
	apAxis[2] := ADR(Axis_2);
	apAxis[3] := ADR(Axis_3);
	bForward := TRUE;
	bBackward := TRUE;
	bFirstRun := FALSE;
END_IF

IF bEnable = FALSE THEN
	bMoveStatus := 2;
END_IF

CASE bMoveStatus OF
	0 :
		bForward := TRUE;
		bBackward := FALSE;
	1 :
		bForward := FALSE;
		bBackward := TRUE;
	2 :
		bForward := FALSE;
		bBackward := FALSE;
END_CASE

FOR iCounter:=0 TO 3 BY 1 DO
	apMC_Power[iCounter](
		Axis:= apAxis[iCounter]^,
		Enable:= TRUE,
		bRegulatorOn:= bEnable,
		bDriveStart:= TRUE,
		Status=> , 
		bRegulatorRealState=> , 
		bDriveStartRealState=> , 
		Busy=> , 
		Error=> , 
		ErrorID=> );
END_FOR

IF bSingleAxisMove = TRUE THEN
	apMC_Jog[iAxisNum](
		Axis:= apAxis[iAxisNum]^, 
		JogForward:= bForward, 
		JogBackward:= bBackward, 
		Velocity:= iVel, 
		Acceleration:= 100, 
		Deceleration:= 100, 
		Jerk:=, 
		Busy=> , 
		CommandAborted=> , 
		Error=> , 
		ErrorId=> );
END_IF

IF bMoveTo = TRUE THEN
	IF bMoveToDone = TRUE THEN
		bMoveTo := FALSE;
	END_IF
	
	apMC_MoveAbsolute[iAxisNum](
		Axis:=apAxis[iAxisNum]^ , 
		Execute:= bMoveTo, 
		Position:= apAxis[iAxisNum]^.fSetPosition + bMoveToLen, 
		Velocity:= iVel, 
		Acceleration:= 10, 
		Deceleration:= 10, 
		Jerk:= 50, 
		Direction:= , 
		Done=> bMoveToDone, 
		Busy=> , 
		CommandAborted=> , 
		Error=> , 
		ErrorID=> );
END_IF

IF bContinusMove = TRUE THEN
	FOR iCounter:=0 TO 3 BY 1 DO
		apMC_Jog[iCounter](
			Axis:= apAxis[iCounter]^, 
			JogForward:= bForward, 
			JogBackward:= bBackward, 
			Velocity:= iVel, 
			Acceleration:= 100, 
			Deceleration:= 100, 
			Jerk:=, 
			Busy=> , 
			CommandAborted=> , 
			Error=> , 
			ErrorId=> );
	END_FOR	
END_IF

IF bSinMove THEN
	lResult := SIN(0.0005 * lSinFreq) * dSinAmpl;
	lSinFreq := lSinFreq + lSinFreqStep;
	
	apAxis[0]^.fSetPosition := apAxis[0]^.fSetPosition + lResult;		//插补下发	
	apAxis[1]^.fSetPosition := apAxis[1]^.fSetPosition + lResult;
	apAxis[2]^.fSetPosition := apAxis[2]^.fSetPosition + lResult;
	apAxis[3]^.fSetPosition := apAxis[3]^.fSetPosition + lResult;

// 	lSum := lSum + 0.002;
// 	IF lSum < 1.0 THEN
// 		apAxis[0]^.fSetPosition := apAxis[0]^.fSetPosition + 0.002;
// 	END_IF

END_IF

adFbPosTest[0] := apAxis[0]^.fActPosition;
adFbPosTest[1] := apAxis[1]^.fActPosition;
adFbPosTest[2] := apAxis[2]^.fActPosition;
adFbPosTest[3] := apAxis[3]^.fActPosition;

FOR iCounter:=0 TO 3 BY 1 DO
	apMC_Reset[iCounter](Axis:=apAxis[iCounter]^, Execute:=bReset, Done=> , Busy=> , Error=> , ErrorID=> );
END_FOR

END_PROGRAM
